// TIA Portal V19 export
VAR_GLOBAL   // PLC tag table "Test6425"
   test1 AT %I0.0 : Bool;
END_VAR
